FUNCTION_BLOCK Room_Ctx_Hmi
VAR_INPUT
	sStatusText				: Str;
	sErrorText				: Str;
	nStatusColor			: Color;
	
	sData					: Str;
	
	bDisable				: BOOL;
	sDisableText			: Str;
	
	bReset					: BOOL;
	bHideReset				: BOOL;
END_VAR
VAR_OUTPUT PERSISTENT
	nTimeout				: UDINT := TIME_TO_UDINT(T#60S);
END_VAR

END_FUNCTION_BLOCK

(* stored: Version 1.1.0.1
   POU Room_Ctx_Hmi: Id {9536c277-9786-455b-b876-b447754e1a8d}, SpecialFunc None *)
